{attribute addProperty BoxType "EL6201-0000-0018"}
{attribute addProperty Id "ASI_Inputs_DeviceAT %I*ASI_Inputs_Device_6E2FC913248310ASI_StatusAT %I*ASI_Status_11283DE6104130ASI_Outputs_DeviceAT %Q*ASI_Outputs_Device_4A17E548248310ASI_ControlAT %Q*ASI_Control_0464DCDE5670WcStateAT %I*WcState_F855686C1620InfoDataAT %I*InfoData_BC63D37F80100"}
{attribute addProperty CRC "2269414939"}
{attribute addProperty SizeInBites "752"}
{attribute addProperty SizeInBytes "94"}
TYPE EL6201_C873A9DB :
STRUCT
	{attribute addProperty Name "ASI_Inputs_Device"}
	ASI_Inputs_Device : ASI_Inputs_Device_6E2FC913;
	{attribute addProperty Name "ASI_Status"}
	ASI_Status : ASI_Status_11283DE6;
	{attribute addProperty Name "ASI_Outputs_Device"}
	ASI_Outputs_Device : ASI_Outputs_Device_4A17E548;
	{attribute addProperty Name "ASI_Control"}
	ASI_Control : ASI_Control_0464DCDE;
	{attribute addProperty Name "WcState"}
	WcState : WcState_F855686C;
	{attribute addProperty Name "InfoData"}
	InfoData : InfoData_BC63D37F;
END_STRUCT
END_TYPE

(* stored: Version 1.2.0.0, ProductVersion 3.1.4024.9
   DUT EL6201_C873A9DB: Id {4dc799d5-9227-4fe2-9012-86100ad973e5} *)
